TYPE ST_PhysicalOutputs :
STRUCT
    bSafetyRunRequest                  : BOOL;
    bSafetyResetRequest                : BOOL;
    bSafetyErrorAcknowledgementRequest : BOOL;
    bAirSupplyEnable                   : BOOL;
    bMainDoorLockRequest               : BOOL;
    bIndexRotatePortA                  : BOOL;
    bIndexStopPortB                    : BOOL;

    // Link to Festo EtherCAT valve-manifold PDOs during commissioning.
    bStation1SupportExtend             : BOOL;
    bStation1SupportRetract            : BOOL;
    bStation2SupportExtend             : BOOL;
    bStation2SupportRetract            : BOOL;
    bStation3SupportExtend             : BOOL;
    bStation3SupportRetract            : BOOL;
	
	bPatchDispenserAir 					: BOOL;
	bPatchVerticalDown 					: BOOL;
	bPatchVerticalUp   					: BOOL;


    // Vision Station / Flipping tooling
    bVisionHorizontalBack              : BOOL;
    bVisionHorizontalFront             : BOOL;
    bVisionVerticalUp                  : BOOL;
    bVisionVerticalDown                : BOOL;
    bVisionLimitOff                    : BOOL;
    bVisionLimitOn                     : BOOL;
    bVisionGripClose                   : BOOL;
    bVisionGripOpen                    : BOOL;
    bVisionRotate0                     : BOOL;
    bVisionRotate180                   : BOOL;

    bHeatStakeHeadLock                 : BOOL;
    bHeatStakeHeadUnlock               : BOOL;
    bHeatStakeHeadDown                 : BOOL;
    bHeatStakeHeadUp                   : BOOL;
    iHeatStakePressureRaw              : INT;

    bLedStart                          : BOOL;
    bLedReset                          : BOOL;
    bStatusIndicatorRed                : BOOL;
    bStatusIndicatorGreen              : BOOL;
    bInternalLight                     : BOOL;
    bNestLight                         : BOOL;
    uiHeatStakePwm1Raw                 : UINT;
    uiHeatStakePwm2Raw                 : UINT;
END_STRUCT
END_TYPE

(* stored: Version 1.1.0.1, ProductVersion 3.1.4026.18
   DUT ST_PhysicalOutputs: Id {c6982397-4202-4d85-945a-2aa8bb403ca0} *)
